% RSLogix 500 project A.RSS, saved by version 8.30.00.16 %
PROJECT "UNTITLED"    % processor: Bul.1763 MicroLogix 1100 Series B %

PROGRAM FILES
  LAD 2   3 rungs

DATA FILES
  O0 OUTPUT  4 elements
  I1 INPUT  6 elements
  S2 STATUS  66 elements
  B3 BINARY  1 elements
  T4 TIMER  1 elements
  C5 COUNTER  1 elements
  R6 CONTROL  1 elements
  N7 INTEGER  1 elements
  F8 FLOAT  1 elements

LADDER 2
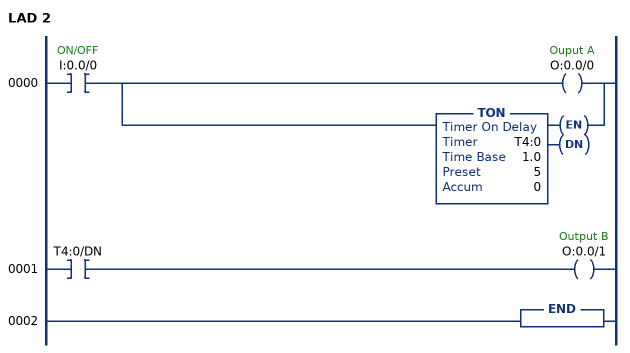
% Rung: 0 %
SOR XIC I:0.0/0 BST OTE O:0.0/0 NXB TON T4:0 1.0 5 0 BND EOR
%   I:0.0/0  "ON/OFF" %
%   O:0.0/0  "Ouput A" %
% Rung: 1 %
SOR XIC T4:0/DN OTE O:0.0/1 EOR
%   O:0.0/1  "Output B" %
% Rung: 2 %
SOR END EOR

OTHER DOCUMENTED ADDRESSES
  I:0.0/1  "OFF"

DATA TABLE (non-zero values as saved)
DATA T4
% .PRE .ACC %
% T4:0 % 5 0
